FUNCTION_BLOCK AdsSocket
VAR_INPUT
END_VAR
VAR_OUTPUT
	//descriptive string for the name of the running program, may or may not be used
	PrgName : STRING;
	
	(*
	AmsNetId should be in the following format for ALL Beckhoff PLCs in the network:
		<area number> . <subarea number (0 for master PLC)> .131.216.1.1
		panel PCs to be assigned 113.174 instead of 131.216
			2.0.131.216.1.1 - Area 2, master controller
			4.3.113.174.1.1 - Area 4, manual station 3 panel PC
	*)
	AmsNetId : T_AmsNetId;
	
	//for now, use ADS port 851 for communication
	AmsPort : T_AmsPort;
END_VAR
VAR_OUTPUT
	receivingData : AdsData;
	sendingData : AdsData;
	
	readBusy : BOOL;
	readError : BOOL;
	readErrorId : UDINT;
	
	writeBusy : BOOL;
	writeError : BOOL;
	writeErrorId : UDINT;
END_VAR
VAR	
	adsWriteSymbol : FB_WriteAdsSymByName;
	adsReadSymbol : FB_ReadAdsSymByName;
END_VAR
VAR
	targetSocket : STRING;
	clearing : BOOL;
END_VAR
(*
TCP-style ADS connection that only writes to a buffer in the recipient's AdsTcpUnit module
*)

//write into the recipient's allocated socket for this system
(*
IF FIND(AmsNetId, '113.174') > 0 THEN //panel PC
	targetSocket := CONCAT('AdsTcp_WinCE.', LocalSocket.PrgName);
ELSE//CX5130+ IPC
	targetSocket := CONCAT('AdsTcp_WinStd.', LocalSocket.PrgName);
END_IF
*)
targetSocket := CONCAT('AdsTcp_WinCE.', LocalSocket.PrgName);
//only toggles if data has contents, otherwise remains false
adsWriteSymbol.bWrite := NOT BufferIsEmpty(sendingData.binaryData) AND NOT adsWriteSymbol.bWrite;
(*
IF NOT BufferIsEmpty(sendingData.binaryData) THEN
	adsWriteSymbol.bWrite := NOT adsWriteSymbol.bWrite;
ELSE
	adsWriteSymbol.bWrite := FALSE;
END_IF 
*)
blocks();

IF NOT adsWriteSymbol.bBusy THEN
	MEMSET(ADR(sendingData), 0, SIZEOF(sendingData));
END_IF

METHOD PRIVATE blocks : BOOL
VAR_INPUT
END_VAR
adsReadSymbol(
	bRead:= , 
	sNetId:= AmsNetId, 
	nPort:= AmsPort, 
	sVarName:= , 
	nDestAddr:= , 
	nLen:= , 
	tTimeout:= , 
	eComMode:= , 
	bClearOnError:= , 
	bBusy=> readBusy, 
	bError=> readError, 
	nErrorId=> readErrorId);
	
adsWriteSymbol(
	bWrite:= , 
	sNetId:= AmsNetId, 
	nPort:= AmsPort, 
	sVarName:= CONCAT(targetSocket, '.receivingData'), 
	nSrcAddr:= ADR(sendingData), 
	nLen:= SIZEOF(sendingData), 
	tTimeout:= , 
	eComMode:= eAdsComModeSecureCom, 
	bBusy=> writeBusy, 
	bError=> writeError, 
	nErrorId=> writeErrorId);
END_METHOD

METHOD send : BOOL
VAR_INPUT
	data : REFERENCE TO AdsData;
END_VAR
sendingData := data;
END_METHOD

END_FUNCTION_BLOCK

(* stored: Version 1.1.0.1, ProductVersion 3.1.4024.11
   POU AdsSocket: Id {9b0b2638-6675-43a4-9f9d-8a56b4ee680d}, SpecialFunc None
   Method blocks: Id {99bfb86b-7d98-4aea-974e-1d1e3d101d3b}
   Method send: Id {6a9cbdb2-3886-45d8-ac84-de738d8e37da} *)
